{attribute addProperty BoxType "APS4322-7000-0017"}
{attribute addProperty Id "CommControlWordAT %Q*UINT16217Data_1AT %Q*UINT16218"}
{attribute addProperty CRC "3518943172"}
{attribute addProperty SizeInBites "32"}
{attribute addProperty SizeInBytes "4"}
TYPE APS_Comm_Outputs_D1BECFC4 :
STRUCT
	{attribute addProperty Name "CommControlWord"}
	CommControlWord AT %Q* : UINT;
	{attribute addProperty Name "Data_1"}
	Data_1 AT %Q* : UINT;
END_STRUCT
END_TYPE

(* stored: Version 1.2.0.0, ProductVersion 3.1.4024.9
   DUT APS_Comm_Outputs_D1BECFC4: Id {d816e885-6252-4fe0-a60c-ddfa17befac2} *)
